# B&R Automation Studio project Lyskryds_i_to_retninger_agdp
Automation Studio 4.8.2.72

## Configuration Config1

### Task classes (Cpu.sw)
```
Cyclic#4:
  Program <- Program.prg
  Program1 <- Program1.prg
  PeerAssesm <- PeerAssesment.prg
  PeerAsses1 <- PeerAssesment1.prg
Binaries: udbdef, FWRules, TCData, sysconf, Role, User, iomap, ashwd, asfw, arconfig, ashwac
Libraries: standard, runtime, astime, asieccon
```

### Hardware
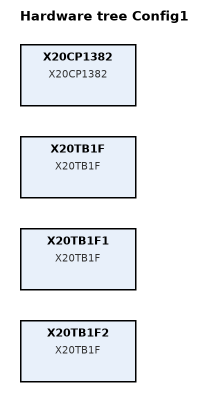
```
X20CP1382 : X20CP1382 v1.10.0.0  [X1 -> X1.SL; X2 -> X2.SL; X3 -> X3.SL]
  Module X1 (Type=X1, Virtual=true, Version=1.10.0.0)
    Connection (Connector=SS1, TargetModule=X20TB1F, TargetConnector=SS)
    Connection (Connector=SL, TargetModule=X20CP1382, TargetConnector=X1)
  Module X2 (Type=X2, Virtual=true, Version=1.10.0.0)
    Connection (Connector=SS1, TargetModule=X20TB1F1, TargetConnector=SS)
    Connection (Connector=SL, TargetModule=X20CP1382, TargetConnector=X2)
  Module X3 (Type=X3, Virtual=true, Version=1.10.0.0)
    Connection (Connector=SS1, TargetModule=X20TB1F2, TargetConnector=SS)
    Connection (Connector=SL, TargetModule=X20CP1382, TargetConnector=X3)
  Connector IF2:
    ActivateDevice = 1
  ConfigurationID = Lyskryds_i_to_retninger_agdp_Config1
  Simulation = 1
X20TB1F : X20TB1F v1.0.0.0
X20TB1F1 : X20TB1F v1.0.0.0
X20TB1F2 : X20TB1F v1.0.0.0
```

## Logical view

### Program Logical/Program (IEC)

#### Types.typ
```iecst
TYPE
	TRAFFICLIGHT :
		(
		RED,
		REDYELLOW,
		YELLOW,
		GREEN
		);
END_TYPE
```

#### Variables.var
```iecst
VAR
	tlight2 : TRAFFICLIGHT;
	tlight1 : TRAFFICLIGHT;
	yellow1 : BOOL;
	green1 : BOOL;
	red1 : BOOL;
	yellow2 : BOOL;
	green2 : BOOL;
	red2 : BOOL;
	timer1 : TON;
	timer2 : TON;
	direction : BOOL;
	old_sensor : BOOL;
	diSensor : BOOL;
	shift : BOOL;
	ready : BOOL;
END_VAR
```

#### Main.st
```iecst
PROGRAM _INIT
	(* Insert code here *)
	ready := TRUE;

END_PROGRAM

PROGRAM _CYCLIC
	// Tilstandsskiftlogik / state change logic
	timer1.IN := TRUE;
	CASE tlight1 OF
		RED:
			timer1.PT := T#2s;
			IF timer1.Q AND direction AND ready THEN
				ready := FALSE;
				tlight1 := REDYELLOW;
				timer1.IN := FALSE;
			END_IF;
		REDYELLOW:
			timer1.PT := T#2s;
			IF timer1.Q AND direction THEN
				tlight1 := GREEN;
				timer1.IN := FALSE;
			END_IF;
		GREEN:
			timer1.PT := T#2s;
			IF timer1.Q AND direction AND shift THEN
				tlight1 := YELLOW;
				timer1.IN := FALSE;
			END_IF;
		YELLOW:
			direction := 0;
			timer1.PT := T#2s;
			IF timer1.Q THEN
				ready := TRUE;
				tlight1 := RED;
				timer1.IN := FALSE;
			END_IF;
	END_CASE
	timer1();

	timer2.IN := TRUE;
	CASE tlight2 OF
		RED:
			timer2.PT := T#2s;
			IF timer2.Q AND NOT(direction) AND ready THEN
				ready := FALSE;
				tlight2 := REDYELLOW;
				timer2.IN := FALSE;
			END_IF;
		REDYELLOW:
			timer2.PT := T#2s;
			IF timer2.Q AND NOT(direction) THEN
				tlight2 := GREEN;
				timer2.IN := FALSE;
			END_IF;
		GREEN:
			timer2.PT := T#2s;
			IF timer2.Q AND NOT(direction) AND shift THEN
				tlight2 := YELLOW;
				timer2.IN := FALSE;
			END_IF;
		YELLOW:
			direction := 1;
			timer2.PT := T#2s;
			IF timer2.Q THEN
				ready := TRUE;
				tlight2 := RED;
				timer2.IN := FALSE;
			END_IF;
	END_CASE
	timer2();

	// OUTPUT LOGIC
	CASE tlight1 OF
		RED:
			red1 := TRUE;
			yellow1 := FALSE;
			green1 := FALSE;
		REDYELLOW:
			red1 := TRUE;
			yellow1 := TRUE;
			green1 := FALSE;
		GREEN:
			red1 := FALSE;
			yellow1 := FALSE;
			green1 := TRUE;
		YELLOW:
			red1 := FALSE;
			yellow1 := TRUE;
			green1 := FALSE;
	END_CASE

	// OUTPUT LOGIC
	CASE tlight2 OF
		RED:
			red2 := TRUE;
			yellow2 := FALSE;
			green2 := FALSE;
		REDYELLOW:
			red2 := TRUE;
			yellow2 := TRUE;
			green2 := FALSE;
		GREEN:
			red2 := FALSE;
			yellow2 := FALSE;
			green2 := TRUE;
		YELLOW:
			red2 := FALSE;
			yellow2 := TRUE;
			green2 := FALSE;
	END_CASE

	shift := NOT old_sensor AND diSensor;
	old_sensor := diSensor;
	IF shift = NOT(diSensor) THEN
		diSensor := FALSE;
	END_IF;

END_PROGRAM

PROGRAM _EXIT
	(* Insert code here *)

END_PROGRAM
```

### Program Logical/Program1 (IEC)

#### Variables.var
```iecst
VAR
	tlight2 : TRAFFICLIGHT;
	tlight1 : TRAFFICLIGHT;
	yellow1 : BOOL;
	green1 : BOOL;
	red1 : BOOL;
	yellow2 : BOOL;
	green2 : BOOL;
	red2 : BOOL;
	timer1 : TON;
	timer2 : TON;
	direction : BOOL;
	diSensor2 : BOOL;
	diSensor1 : BOOL;
	ready : BOOL;
END_VAR
```

#### Main.st
```iecst
PROGRAM _INIT
	(* Insert code here *)
	ready := TRUE;

END_PROGRAM

PROGRAM _CYCLIC
	// Tilstandsskiftlogik / state change logic
	timer1.IN := TRUE;
	CASE tlight1 OF
		RED:
			timer1.PT := T#2s;
			IF timer1.Q AND direction AND ready THEN
				ready := FALSE;
				tlight1 := REDYELLOW;
				timer1.IN := FALSE;
			END_IF;
		REDYELLOW:
			timer1.PT := T#2s;
			IF timer1.Q AND direction THEN
				tlight1 := GREEN;
				timer1.IN := FALSE;
			END_IF;
		GREEN:
			timer1.PT := T#2s;
			IF timer1.Q AND direction AND diSensor2 THEN
				tlight1 := YELLOW;
				timer1.IN := FALSE;
			END_IF;
		YELLOW:
			direction := 0;
			timer1.PT := T#2s;
			IF timer1.Q THEN
				ready := TRUE;
				tlight1 := RED;
				timer1.IN := FALSE;
			END_IF;
	END_CASE
	timer1();

	timer2.IN := TRUE;
	CASE tlight2 OF
		RED:
			timer2.PT := T#2s;
			IF timer2.Q AND NOT(direction) AND ready THEN
				ready := FALSE;
				tlight2 := REDYELLOW;
				timer2.IN := FALSE;
			END_IF;
		REDYELLOW:
			timer2.PT := T#2s;
			IF timer2.Q AND NOT(direction) THEN
				tlight2 := GREEN;
				timer2.IN := FALSE;
			END_IF;
		GREEN:
			timer2.PT := T#2s;
			IF timer2.Q AND NOT(direction) AND diSensor1 THEN
				tlight2 := YELLOW;
				timer2.IN := FALSE;
			END_IF;
		YELLOW:
			direction := 1;
			timer2.PT := T#2s;
			IF timer2.Q THEN
				ready := TRUE;
				tlight2 := RED;
				timer2.IN := FALSE;
			END_IF;
	END_CASE
	timer2();

	// OUTPUT LOGIC
	CASE tlight1 OF
		RED:
			red1 := TRUE;
			yellow1 := FALSE;
			green1 := FALSE;
		REDYELLOW:
			red1 := TRUE;
			yellow1 := TRUE;
			green1 := FALSE;
		GREEN:
			red1 := FALSE;
			yellow1 := FALSE;
			green1 := TRUE;
		YELLOW:
			red1 := FALSE;
			yellow1 := TRUE;
			green1 := FALSE;
	END_CASE

	// OUTPUT LOGIC
	CASE tlight2 OF
		RED:
			red2 := TRUE;
			yellow2 := FALSE;
			green2 := FALSE;
		REDYELLOW:
			red2 := TRUE;
			yellow2 := TRUE;
			green2 := FALSE;
		GREEN:
			red2 := FALSE;
			yellow2 := FALSE;
			green2 := TRUE;
		YELLOW:
			red2 := FALSE;
			yellow2 := TRUE;
			green2 := FALSE;
	END_CASE

END_PROGRAM

PROGRAM _EXIT
	(* Insert code here *)

END_PROGRAM
```

### Program Logical/PeerAssesment (IEC)

#### Types.typ
```iecst
TYPE
	TRAFFIC_LIGHT :
		(
		TRAFFIC_LIGHT_GREEN,
		TRAFFIC_LIGHT_YELLOW,
		TRAFFIC_LIGHT_REDYELLOW,
		TRAFFIC_LIGHT_RED
		);
END_TYPE
```

#### Variables.var
```iecst
VAR
	doGreen2 : BOOL;
	doYellow2 : BOOL;
	doRed2 : BOOL;
	trafficst : TRAFFIC_LIGHT;
	shift : BOOL;
	doRed : BOOL;
	doYellow : BOOL;
	doGreen : BOOL;
	timer : TON;
	traffic2st : TRAFFIC_LIGHT;
END_VAR
```

#### Main.st
```iecst
PROGRAM _INIT
	(* Insert code here *)
 trafficst := TRAFFIC_LIGHT_RED;
END_PROGRAM

PROGRAM _CYCLIC
//Når der er grønt i en retning skal modsatte retning have rødt
//Når der er gul i en retning skal der være rødt i modsat retning
//Når der skiftes fra gul til rød i en retning skal der skiftes til gulrød i anden retning
//Der skal anvendes timer til at have 2 sekunder mellem farveskift.
//Der skal anvendes et signal til at signalere start for hvornår, der skal skiftes fra grøn til gul

	(* Insert code here *)
	// Tilstandsskift

	CASE trafficst OF
		TRAFFIC_LIGHT_RED:
			IF (traffic2st = TRAFFIC_LIGHT_RED) THEN
				trafficst := TRAFFIC_LIGHT_REDYELLOW;
			END_IF

		TRAFFIC_LIGHT_REDYELLOW:
			timer(IN := TRUE, PT := T#2000ms);
			IF timer.Q THEN
				timer(IN := FALSE);
				trafficst := TRAFFIC_LIGHT_GREEN;
			END_IF

		TRAFFIC_LIGHT_YELLOW:
			timer(IN := TRUE, PT := T#2000ms);
			IF timer.Q THEN
				timer(IN := FALSE);
				trafficst := TRAFFIC_LIGHT_RED;
			END_IF

		TRAFFIC_LIGHT_GREEN:
			timer(IN := TRUE, PT := T#2000ms);
			IF timer.Q AND shift THEN
				timer(IN := FALSE);
				trafficst := TRAFFIC_LIGHT_YELLOW;
			END_IF

	END_CASE

	CASE traffic2st OF
		TRAFFIC_LIGHT_RED:
			IF (trafficst = TRAFFIC_LIGHT_RED) THEN
				traffic2st := TRAFFIC_LIGHT_REDYELLOW;
			END_IF

		TRAFFIC_LIGHT_REDYELLOW:
			timer(IN := TRUE, PT := T#2000ms);
			IF timer.Q THEN
				timer(IN := FALSE);
				traffic2st := TRAFFIC_LIGHT_GREEN;
			END_IF

		TRAFFIC_LIGHT_YELLOW:
			timer(IN := TRUE, PT := T#2000ms);
			IF timer.Q THEN
				timer(IN := FALSE);
				traffic2st := TRAFFIC_LIGHT_RED;
			END_IF

		TRAFFIC_LIGHT_GREEN:
			timer(IN := TRUE, PT := T#2000ms);
			IF timer.Q AND shift THEN
				timer(IN := FALSE);
				traffic2st := TRAFFIC_LIGHT_YELLOW;
			END_IF

		END_CASE

	// Output logic
	CASE trafficst OF
		TRAFFIC_LIGHT_RED:
			doRed := TRUE;
			doYellow := FALSE;
			doGreen := FALSE;

		TRAFFIC_LIGHT_REDYELLOW:
			doRed := TRUE;
			doYellow := TRUE;
			doGreen := FALSE;

		TRAFFIC_LIGHT_YELLOW:
			doRed := FALSE;
			doYellow := TRUE;
			doGreen := FALSE;

		TRAFFIC_LIGHT_GREEN:
			doRed := FALSE;
			doYellow := FALSE;
			doGreen := TRUE;
	END_CASE

	CASE traffic2st OF
		TRAFFIC_LIGHT_RED:
			doRed2 := TRUE;
			doYellow2 := FALSE;
			doGreen2 := FALSE;

		TRAFFIC_LIGHT_REDYELLOW:
			doRed2 := TRUE;
			doYellow2 := TRUE;
			doGreen2 := FALSE;

		TRAFFIC_LIGHT_YELLOW:
			doRed2 := FALSE;
			doYellow2 := TRUE;
			doGreen2 := FALSE;

		TRAFFIC_LIGHT_GREEN:
			doRed2 := FALSE;
			doYellow2 := FALSE;
			doGreen2 := TRUE;

	END_CASE

END_PROGRAM

PROGRAM _EXIT
	(* Insert code here *)

END_PROGRAM
```

### Program Logical/PeerAssesment1 (IEC)

#### Types.typ
```iecst
TYPE
	TRAFFIC_LIGHT :
		(
		TRAFFIC_LIGHT1_RED,
		TRAFFIC_LIGHT2_RED,
		TRAFFIC_LIGHT1_REDYELLOW,
		TRAFFIC_LIGHT2_REDYELLOW,
		TRAFFIC_LIGHT1_YELLOW,
		TRAFFIC_LIGHT2_YELLOW,
		TRAFFIC_LIGHT1_GREEN,
		TRAFFIC_LIGHT2_GREEN
		);
END_TYPE
```

#### Variables.var
```iecst
VAR
	shift : BOOL;
	trafficst : TRAFFIC_LIGHT;
	timer : TON;
	doGreen : BOOL;
	doYellow : BOOL;
	doRed : BOOL;
	doRed2 : BOOL;
	doYellow2 : BOOL;
	doGreen2 : BOOL;
END_VAR
```

#### Main.st
```iecst
PROGRAM _INIT
	(* Insert code here *)
END_PROGRAM

PROGRAM _CYCLIC

	// Tilstandsskift

	CASE trafficst OF
		TRAFFIC_LIGHT1_RED:
			timer(IN := TRUE, PT := T#2000ms);
			IF timer.Q AND shift THEN
				timer(IN := FALSE);
				trafficst := TRAFFIC_LIGHT1_REDYELLOW;
			END_IF

		TRAFFIC_LIGHT1_GREEN:
			timer(IN := TRUE, PT := T#2000ms);
			IF timer.Q AND shift THEN
				timer(IN := FALSE);
				trafficst := TRAFFIC_LIGHT1_YELLOW;
			END_IF

		TRAFFIC_LIGHT1_REDYELLOW:
			timer(IN := TRUE, PT := T#2000ms);
			IF timer.Q THEN
				timer(IN := FALSE);
				trafficst := TRAFFIC_LIGHT1_GREEN;
			END_IF

		TRAFFIC_LIGHT1_YELLOW:
			timer(IN := TRUE, PT := T#2000ms);
			IF timer.Q THEN
				timer(IN := FALSE);
				trafficst := TRAFFIC_LIGHT1_RED;
				trafficst := TRAFFIC_LIGHT2_REDYELLOW;
			END_IF

		TRAFFIC_LIGHT2_RED:
			timer(IN := TRUE, PT := T#2000ms);
			IF timer.Q AND shift THEN
				timer(IN := FALSE);
				trafficst := TRAFFIC_LIGHT2_REDYELLOW;
			END_IF

		TRAFFIC_LIGHT2_GREEN:
			timer(IN := TRUE, PT := T#2000ms);
			IF timer.Q AND shift THEN
				timer(IN := FALSE);
				trafficst := TRAFFIC_LIGHT2_YELLOW;
			END_IF

		TRAFFIC_LIGHT2_REDYELLOW:
			timer(IN := TRUE, PT := T#2000ms);
			IF timer.Q THEN
				timer(IN := FALSE);
				trafficst := TRAFFIC_LIGHT2_GREEN;
			END_IF

		TRAFFIC_LIGHT2_YELLOW:
			timer(IN := TRUE, PT := T#2000ms);
			IF timer.Q THEN
				timer(IN := FALSE);
				trafficst := TRAFFIC_LIGHT2_RED;
				trafficst := TRAFFIC_LIGHT1_REDYELLOW;
			END_IF

	END_CASE

	// Output logic
	CASE trafficst OF
		TRAFFIC_LIGHT1_RED:
			doRed := TRUE;
			doYellow := FALSE;
			doGreen := FALSE;
			doRed2 := FALSE;
			doYellow2 := FALSE;
			doGreen2 := TRUE;

		TRAFFIC_LIGHT1_REDYELLOW:
			doRed := TRUE;
			doYellow := TRUE;
			doGreen := FALSE;
			doRed2 := TRUE;
			doYellow2 := FALSE;
			doGreen2 := FALSE;

		TRAFFIC_LIGHT1_YELLOW:
			doRed := FALSE;
			doYellow := TRUE;
			doGreen := FALSE;
			doRed2 := TRUE;
			doYellow2 := FALSE;
			doGreen2 := FALSE;

		TRAFFIC_LIGHT1_GREEN:
			doRed := FALSE;
			doYellow := FALSE;
			doGreen := TRUE;
			doRed2 := TRUE;
			doYellow2 := FALSE;
			doGreen2 := FALSE;

		TRAFFIC_LIGHT2_RED:
			doRed2 := TRUE;
			doYellow2 := FALSE;
			doGreen2 := FALSE;
			doRed := FALSE;
			doYellow := FALSE;
			doGreen := TRUE;

		TRAFFIC_LIGHT2_REDYELLOW:
			doRed2 := TRUE;
			doYellow2 := TRUE;
			doGreen2 := FALSE;
			doRed := TRUE;
			doYellow := FALSE;
			doGreen := FALSE;

		TRAFFIC_LIGHT2_YELLOW:
			doRed2 := FALSE;
			doYellow2 := TRUE;
			doGreen2 := FALSE;
			doRed := TRUE;
			doYellow := FALSE;
			doGreen := FALSE;

		TRAFFIC_LIGHT2_GREEN:
			doRed2 := FALSE;
			doYellow2 := FALSE;
			doGreen2 := TRUE;
			doRed := TRUE;
			doYellow := FALSE;
			doGreen := FALSE;
	END_CASE

END_PROGRAM

PROGRAM _EXIT
	(* Insert code here *)

END_PROGRAM
```

Listed in the project but not available here: Logical/Global.typ, Logical/Global.var, Logical/Libraries
